{attribute clr [Container(Layout.Stack)]}
{attribute clr [Group(Layout.GroupBox)]}
{attribute addProperty PreviousPort "Unknown"}
TYPE EtcSlaveTerminalBase :
STRUCT
END_STRUCT
END_TYPE

(* stored: Version 1.1.0.1, ProductVersion 3.1.4024.9
   DUT EtcSlaveTerminalBase: Id {b93e26cd-5441-0782-1f60-5eb68061b724} *)
